{attribute 'qualified_only'}
//Axis day 2 training
VAR_GLOBAL
	Axis_servoA : AXIS_REF;
	Axis_servoB : AXIS_REF;
	Axis_servoVirtual : AXIS_REF;
	Axis_servo : AXIS_REF; 
END_VAR

(* stored: Version 1.1.0.1, ProductVersion 3.1.4024.12
   GVL GVL: Id {1681d69f-05d1-44d7-a747-dbb565223030} *)
